///Checks if the returned HRESULT is success and busy
FUNCTION Busy : BOOL
VAR_INPUT
    hr : HRESULT;
END_VAR
VAR
END_VAR

Busy := (hr = HResultSuccess.Busy);

END_FUNCTION

(* stored: Version 1.1.0.1, ProductVersion 3.1.4020.12
   POU Busy: Id {bb15b117-3bbc-4dce-a8e4-e5608e416082}, SpecialFunc None *)
